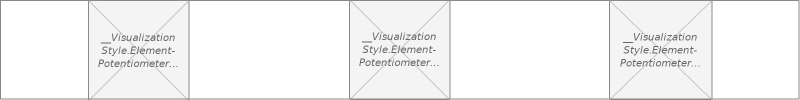
VISUALIZATION Nav_1  // 800x100
    Image (609,0 103x100)
        OnMouseDown: change screen: Charge_Velocity_Distance
    Image (88,0 101x101)
        OnMouseDown: change screen: Safty_Zones_and_Modes
    Image (349,-1 101x101)
        OnMouseDown: change screen: MainScreen
END_VISUALIZATION

(* stored: Version 1.1.0.1, ProductVersion 3.1.4024.12
   Visu Nav_1: Id {82976a8c-135d-4430-8d32-84095567d3ce} *)
